DATA_BLOCK "DB_SequenceStation"
{ S7_Optimized_Access := 'TRUE' }
VERSION : 0.1
NON_RETAIN
"FB_SequenceStation"
BEGIN
END_DATA_BLOCK
